Staubli VAL3: getdWordAt.pgx

public program getDwordAt(num x_nByteIndex, num& x_nBuffer[], num& x_nRes)
begin

  x_nRes=x_nBuffer[x_nByteIndex]*power(2,24)+x_nBuffer[x_nByteIndex+1]*power(2,16)+x_nBuffer[x_nByteIndex+2]*power(2,8)+x_nBuffer[x_nByteIndex+3]

end
